(* IEC 61131-3 sources: Std_PalletMover/Class/HalBmsMastervoltinterface, 1 file *)

(* ---- HalBmsMastervoltinterface.st ---- *)
(*!
<Class
	Name               = "HalBmsMastervoltinterface"
	Revision           = "0.0"
	RealtimeTask       = "false"
	CyclicTask         = "false"
	BackgroundTask     = "false"
	Sigmatek           = "false"
	OSInterface        = "false"
	HighPriority       = "false"
	Automatic          = "false"
	UpdateMode         = "Prescan"
	SharedCommandTable = "true"
	Objectsize         = "(840,120)">
	<Channels>
		<Client Name="ToBmsMastervolt" Required="true" Internal="false"/>
	</Channels>
	<Network Name="HalBmsMastervoltinterface">
		<!-- List of Components in this network -->
		<Components>
			<Object
				Name       = "_base"
				Class      = "I_Bms"
				Position   = "(218,120)"
				Visualized = "false">
				<Channels>
					<Server Name="ClassSvr"/>
				</Channels>
			</Object>
		</Components>
		<Comments>
		</Comments>
		<!-- List of Connections in this network -->
		<Connections>
			<Connection Source="this.ClassSvr" Destination="_base.ClassSvr" Vertices="(1246,210),(1074,210),"/>
		</Connections>
		<!-- Headerfiles -->
		<Options>
		</Options>
	</Network>
</Class>
*)
#pragma using I_Bms

HalBmsMastervoltinterface : CLASS
: I_Bms
  //Servers:
  //Clients:
	ToBmsMastervolt 	: CltChCmd_HAL_BMS_MasterVolt;
  //Variables:
  //Functions:
  //Tables:
	FUNCTION @STD
		VAR_OUTPUT
			ret_code	: CONFSTATES;
		END_VAR;
	FUNCTION GLOBAL TAB @CT_;
END_CLASS;

#pragma usingLtd HAL_BMS_MasterVolt
